Staubli VAL3: waitCharOnSk.pgx

program waitCharOnSk(string x_sCharacter (dimensions=1))
  local num l_nAsciiCode
  local string l_sCharRead
begin
  // This program reads character by character on the socket until
  //  it finds a specific character. The socket must be a socket
  //  server with timeout=0
  //
  // Input Param
  //  x_sCharacter : Character to find
  //
  // Output Param
  //  none         :
  //
  //----------------------------------------------------------------
  //
  l_sCharRead=""
  //
  // Read character by character until finds specific character
  while l_sCharRead!=x_sCharacter
    // Reads one character from socket
    sioGet(skFromRobot,l_nAsciiCode)
    l_sCharRead=chr(l_nAsciiCode)
  endWhile
  //
end
